{attribute 'qualified_only'}
VAR_GLOBAL
	Err  : BOOL;
END_VAR

(* stored: Version 1.1.0.1
   GVL Err: Id {756d2f22-c434-4cd8-8883-4ebf4fab2410} *)
